// SIMATIC S7-200 project (STEP 7-Micro/WIN), CPU 222 REL 01.22

ORGANIZATION_BLOCK PRINCIPAL:OB1
TITLE=COMENTARIOS DEL PROGRAMA
BEGIN
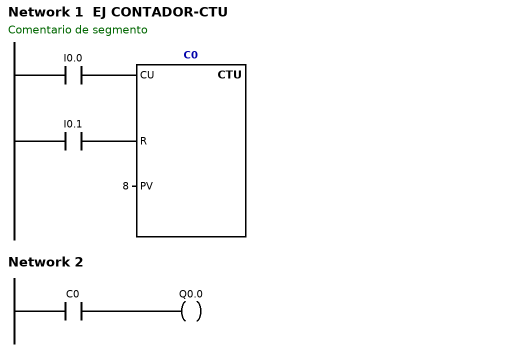
Network 1 // EJ CONTADOR-CTU

// Comentario de segmento
// (network saved uncompiled; LAD cells follow)
// row 0: c0 -| |- I0.0  c1 [CTU C0 CU:=power@row0, R:=power@row1, PV:=8]
// row 1: c0 -| |- I0.1  c1 [box]
// row 2: c1 [box]
Network 2
// (network saved uncompiled; LAD cells follow)
// row 0: c0 -| |- C0  c1 -( ) Q0.0
END_ORGANIZATION_BLOCK
